// TwinCAT 3 PLC project PLC
// ProgramVersion: 3.1.4026.22
// libraries:
//   Tc2_MC2, * (Beckhoff Automation GmbH)
//   Tc2_Standard, * (Beckhoff Automation GmbH)
//   Tc2_System, * (Beckhoff Automation GmbH)
//   Tc3_Module, * (Beckhoff Automation GmbH)
// project tree:
//   DUTs/ E_ControlMode.TcDUT, ST_MotorParameters.TcDUT (not stored)
//   GVLs/ GVL_MotorControl.TcGVL, GVL_Safety.TcGVL
//   / PlcTask.TcTTO
//   POUs/ FB_MotorControl.TcPOU (not stored), MAIN.TcPOU (not stored)
// real-time tasks:
//   TASK PlcTask: cycle T#10ms, priority 20, ADS port 350
// motion (NC):
//   TASK NC-Task 1 SAF: cycle T#2ms, priority 4, ADS port 501
//   TASK NC-Task 1 SVB: cycle T#10ms, priority 8, ADS port 511
//   AXIS Axis 1 (id 1)
//     Dynamic: Acceleration=2545.9695, Deceleration=2545.9695, Jerk=7637.9085
//     Velo: RefSearch=16.97313, RefSync=16.97313, SlowManual=84.86565, FastManual=509.1939, Fast=1697.313, Maximum=1697.313
//     OtherSettings: AllowMotionCmdToSlave=true
//     encoder EncType=19
//       EncPara: ScaleFactorNumerator=60, ScaleFactorDenominator=1048576, MaxCount=#xffffffff
//     drive DrvType=16
//       DrvPara: MaxCount=#xffffffff, DriveControlDWord=#x00020100
//         Analog: VeloReferenz=1867.0443, VeloScale=32, TorqueSetpointScale=10, ScaleFactorActTorque=0.1
//         TimeComp: TaskDelayCycles=1
//     controller CtrType=1
//       CtrPara: PriorControlFactor=1
//         PosDiffControl: Enable=false, Time=1
//         Observer: BandWidth=20
//   AXIS Axis 2 (id 2)
//     Dynamic: Acceleration=2545.9695, Deceleration=2545.9695, Jerk=7637.9085
//     Velo: RefSearch=16.97313, RefSync=16.97313, SlowManual=84.86565, FastManual=509.1939, Fast=1697.313, Maximum=1697.313
//     OtherSettings: AllowMotionCmdToSlave=true
//     encoder EncType=19
//       EncPara: ScaleFactorNumerator=60, ScaleFactorDenominator=1048576, MaxCount=#xffffffff
//     drive DrvType=16
//       DrvPara: MaxCount=#xffffffff, DriveControlDWord=#x00020100
//         Analog: VeloReferenz=1867.0443, VeloScale=32, TorqueSetpointScale=10, ScaleFactorActTorque=0.1
//         TimeComp: TaskDelayCycles=1
//     controller CtrType=1
//       CtrPara: PriorControlFactor=1
//         PosDiffControl: Enable=false
//         Observer: BandWidth=20
//   AXIS Axis 3 (id 3)
//     Dynamic: Acceleration=2545.9695, Deceleration=2545.9695, Jerk=7637.9085
//     Velo: RefSearch=16.97313, RefSync=16.97313, SlowManual=84.86565, FastManual=509.1939, Fast=1697.313, Maximum=1697.313
//     OtherSettings: AllowMotionCmdToSlave=true
//     encoder EncType=19
//       EncPara: ScaleFactorNumerator=60, ScaleFactorDenominator=1048576, MaxCount=#xffffffff
//     drive DrvType=16
//       DrvPara: MaxCount=#xffffffff, DriveControlDWord=#x00020100
//         Analog: VeloReferenz=1867.0443, VeloScale=32, TorqueSetpointScale=10, ScaleFactorActTorque=0.1
//         TimeComp: TaskDelayCycles=1
//     controller CtrType=1
//       CtrPara: PriorControlFactor=1
//         PosDiffControl: Enable=false
//         Observer: BandWidth=20
// I/O:
//   DEVICE Device 1 (EtherCAT), AmsNetId 5.148.118.242.2.1
//     Term 1 (EK1200) [EK1200-5000 EtherCAT Power supply (2A E-Bus)]
//       Term 2 (EL2008) [EL2008 8Ch. Dig. Output 24V, 0.5A]
//       Term 3 (EL1008) [EL1008 8Ch. Dig. Input 24V, 3ms]
//       Term 4 (EL2911) [EL2911, Potential supply terminal (10 A) with 4 Ch. Safety Inputs, TwinSAFE]
//         modules: Module 2 (FSOUT), Module 3 (DEVICEIO), Module 4 (FSLOGIC)
//       Term 5 (EK1122) [EK1122 2 port EtherCAT junction]
//         Term 6 (EK1100) [EK1100 EtherCAT Coupler (2A E-Bus)]
//           Term 7 (EL7062) [EL7062-0000 2Ch. Stepper motor output stage (48V, 3A)]
//             startup 28688:3 := 08 // DRV Outputs Ch.1 / Modes of operation
//             startup 28688:16 := FF7F // DRV Outputs Ch.1 / Positive torque limit value
//             startup 28688:17 := FF7F // DRV Outputs Ch.1 / Negative torque limit value
//             startup 32784:87 := 64 // DRV Amplifier Settings Ch.1 / Position loop velocity feed forward gain
//             startup 32784:109 := 64000000 // DRV Amplifier Settings Ch.1 / Torque feed forward gain
//             startup 32785:52 := 90060000 // DRV Motor Settings Ch.1 / Configured motor current
//             startup 32784:19 := 3600 // DRV Amplifier Settings Ch.1 / Current loop proportional gain
//             startup 32784:18 := 1100 // DRV Amplifier Settings Ch.1 / Current loop integral time
//             startup 32784:21 := 1C000000 // DRV Amplifier Settings Ch.1 / Velocity loop proportional gain
//             startup 32784:20 := 96000000 // DRV Amplifier Settings Ch.1 / Velocity loop integral time
//             startup 28944:3 := 08 // DRV Outputs Ch.2 / Modes of operation
//             startup 28944:16 := FF7F // DRV Outputs Ch.2 / Positive torque limit value
//             startup 28944:17 := FF7F // DRV Outputs Ch.2 / Negative torque limit value
//             startup 33040:87 := 64 // DRV Amplifier Settings Ch.2 / Position loop velocity feed forward gain
//             startup 33040:109 := 64000000 // DRV Amplifier Settings Ch.2 / Torque feed forward gain
//             startup 33041:52 := 90060000 // DRV Motor Settings Ch.2 / Configured motor current
//             startup 33040:19 := 3600 // DRV Amplifier Settings Ch.2 / Current loop proportional gain
//             startup 33040:18 := 1100 // DRV Amplifier Settings Ch.2 / Current loop integral time
//             startup 33040:21 := 1C000000 // DRV Amplifier Settings Ch.2 / Velocity loop proportional gain
//             startup 33040:20 := 96000000 // DRV Amplifier Settings Ch.2 / Velocity loop integral time
//           Term 8 (EL7062) [EL7062-0000 2Ch. Stepper motor output stage (48V, 3A)]
//             startup 28688:3 := 08 // DRV Outputs Ch.1 / Modes of operation
//             startup 28688:16 := FF7F // DRV Outputs Ch.1 / Positive torque limit value
//             startup 28688:17 := FF7F // DRV Outputs Ch.1 / Negative torque limit value
//             startup 32784:87 := 64 // DRV Amplifier Settings Ch.1 / Position loop velocity feed forward gain
//             startup 32784:109 := 64000000 // DRV Amplifier Settings Ch.1 / Torque feed forward gain
//             startup 32785:52 := 90060000 // DRV Motor Settings Ch.1 / Configured motor current
//             startup 32784:19 := 3600 // DRV Amplifier Settings Ch.1 / Current loop proportional gain
//             startup 32784:18 := 1100 // DRV Amplifier Settings Ch.1 / Current loop integral time
//             startup 32784:21 := 1C000000 // DRV Amplifier Settings Ch.1 / Velocity loop proportional gain
//             startup 32784:20 := 96000000 // DRV Amplifier Settings Ch.1 / Velocity loop integral time
//           Term 9 (EL9011) [EL9011 End Terminal]
// variable links:
//   NC-Task 1 SAF/Axes/Axis 1 <-> Device 1 (EtherCAT)/Term 1 (EK1200)/Term 5 (EK1122)/Term 6 (EK1100)/Term 7 (EL7062)
//     Drive/Inputs/In/nDataIn1 <-> DRV Following error actual value Channel 1/Following error actual value
//     Drive/Inputs/In/nDcOutputTime <-> InfoData/DcOutputShift
//     Drive/Inputs/In/nState1 <-> DRV Statusword Channel 1/Statusword
//     Drive/Inputs/In/nState2 <-> DRV Statusword Channel 1/Statusword @bit 8
//     Drive/Inputs/In/nState4 @bit 1 <-> WcState/InputToggle
//     Drive/Inputs/In/nState4 <-> WcState/WcState
//     Drive/Outputs/Out/nCtrl1 <-> DRV Controlword Channel 1/Controlword
//     Drive/Outputs/Out/nCtrl2 <-> DRV Controlword Channel 1/Controlword @bit 8
//     Drive/Outputs/Out/nDataOut1 <-> DRV Target position Channel 1/Target position
//     Enc/Inputs/In/nDataIn1 <-> FB Position Channel 1/Position
//     Enc/Inputs/In/nDcInputTime <-> InfoData/DcInputShift
//     Enc/Inputs/In/nState4 @bit 1 <-> WcState/InputToggle
//     Enc/Inputs/In/nState4 <-> WcState/WcState
//   NC-Task 1 SAF/Axes/Axis 2 <-> Device 1 (EtherCAT)/Term 1 (EK1200)/Term 5 (EK1122)/Term 6 (EK1100)/Term 7 (EL7062)
//     Drive/Inputs/In/nDataIn1 <-> DRV Following error actual value Channel 2/Following error actual value
//     Drive/Inputs/In/nDcOutputTime <-> InfoData/DcOutputShift
//     Drive/Inputs/In/nState1 <-> DRV Statusword Channel 2/Statusword
//     Drive/Inputs/In/nState2 <-> DRV Statusword Channel 2/Statusword @bit 8
//     Drive/Inputs/In/nState4 @bit 1 <-> WcState/InputToggle
//     Drive/Inputs/In/nState4 <-> WcState/WcState
//     Drive/Outputs/Out/nCtrl1 <-> DRV Controlword Channel 2/Controlword
//     Drive/Outputs/Out/nCtrl2 <-> DRV Controlword Channel 2/Controlword @bit 8
//     Drive/Outputs/Out/nDataOut1 <-> DRV Target position Channel 2/Target position
//     Enc/Inputs/In/nDataIn1 <-> FB Position Channel 2/Position
//     Enc/Inputs/In/nDcInputTime <-> InfoData/DcInputShift
//     Enc/Inputs/In/nState4 @bit 1 <-> WcState/InputToggle
//     Enc/Inputs/In/nState4 <-> WcState/WcState
//   NC-Task 1 SAF/Axes/Axis 3 <-> Device 1 (EtherCAT)/Term 1 (EK1200)/Term 5 (EK1122)/Term 6 (EK1100)/Term 8 (EL7062)
//     Drive/Inputs/In/nDataIn1 <-> DRV Following error actual value Channel 1/Following error actual value
//     Drive/Inputs/In/nDcOutputTime <-> InfoData/DcOutputShift
//     Drive/Inputs/In/nState1 <-> DRV Statusword Channel 1/Statusword
//     Drive/Inputs/In/nState2 <-> DRV Statusword Channel 1/Statusword @bit 8
//     Drive/Inputs/In/nState4 @bit 1 <-> WcState/InputToggle
//     Drive/Inputs/In/nState4 <-> WcState/WcState
//     Drive/Outputs/Out/nCtrl1 <-> DRV Controlword Channel 1/Controlword
//     Drive/Outputs/Out/nCtrl2 <-> DRV Controlword Channel 1/Controlword @bit 8
//     Drive/Outputs/Out/nDataOut1 <-> DRV Target position Channel 1/Target position
//     Enc/Inputs/In/nDataIn1 <-> FB Position Channel 1/Position
//     Enc/Inputs/In/nDcInputTime <-> InfoData/DcInputShift
//     Enc/Inputs/In/nState4 @bit 1 <-> WcState/InputToggle
//     Enc/Inputs/In/nState4 <-> WcState/WcState
//   PLC/PLC Instance <-> Device 1 (EtherCAT)/Term 1 (EK1200)/Term 2 (EL2008)
//     PlcTask Outputs/MAIN.greenLight <-> Channel 1/Output
//     PlcTask Outputs/MAIN.orangeLight <-> Channel 2/Output
//     PlcTask Outputs/MAIN.redLight <-> Channel 3/Output
//   PLC/PLC Instance <-> Device 1 (EtherCAT)/Term 1 (EK1200)/Term 3 (EL1008)
//     PlcTask Inputs/MAIN.sw1 <-> Channel 1/Input
//     PlcTask Inputs/MAIN.sw2 <-> Channel 2/Input
//     PlcTask Inputs/MAIN.sw3 <-> Channel 3/Input
//   PLC/PLC Instance <-> Device 1 (EtherCAT)/Term 1 (EK1200)/Term 4 (EL2911)
//     PlcTask Inputs/GVL_Safety.SafetyOutput <-> StandardInputs/TwinSafeGroup1.Output_4
//     PlcTask Outputs/GVL_Safety.SafetyErrAck <-> StandardOutputs/TwinSafeGroup1.ErrorAcknowledgement_1
//     PlcTask Outputs/GVL_Safety.SafetyRestart <-> StandardOutputs/TwinSafeGroup1.Restart_5
//     PlcTask Outputs/GVL_Safety.SafetyRun <-> StandardOutputs/TwinSafeGroup1.Run_2
//   PLC/PLC Instance <-> NC-Task 1 SAF/Axes/Axis 1
//     PlcTask Inputs/MAIN.motor[1].axis.NcToPlc <-> Outputs/ToPlc
//     PlcTask Outputs/MAIN.motor[1].axis.PlcToNc <-> Inputs/FromPlc
//   PLC/PLC Instance <-> NC-Task 1 SAF/Axes/Axis 2
//     PlcTask Inputs/MAIN.motor[2].axis.NcToPlc <-> Outputs/ToPlc
//     PlcTask Outputs/MAIN.motor[2].axis.PlcToNc <-> Inputs/FromPlc
//   PLC/PLC Instance <-> NC-Task 1 SAF/Axes/Axis 3
//     PlcTask Inputs/MAIN.motor[3].axis.NcToPlc <-> Outputs/ToPlc
//     PlcTask Outputs/MAIN.motor[3].axis.PlcToNc <-> Inputs/FromPlc

CONFIGURATION PLC
    RESOURCE PLC ON TwinCAT3
        TASK PlcTask(INTERVAL := T#10ms, PRIORITY := 20);
        PROGRAM MAIN WITH PlcTask : MAIN;
    END_RESOURCE
END_CONFIGURATION

// ---- DUTs/E_ControlMode.TcDUT
{attribute 'qualified_only'}
{attribute 'strict'}
TYPE E_ControlMode :
(
	POSITION := 0,
	VELOCITY := 1
);
END_TYPE

// ---- GVLs/GVL_MotorControl.TcGVL
{attribute 'qualified_only'}
VAR_GLOBAL CONSTANT
	CNUM_AXIS : INT := 3;
END_VAR

// ---- GVLs/GVL_Safety.TcGVL
{attribute 'qualified_only'}
VAR_GLOBAL
	SafetyRun AT %Q* : BOOL;
	SafetyRestart AT %Q* : BOOL;
	SafetyErrAck AT %Q* : BOOL;
	SafetyOutput AT %I* : BOOL; 
END_VAR
